FUNCTION_BLOCK SERVICE_INFO_JSON_DESERIALIZE (* Composite Function Block Type *)
  (* Standard: 61499-2 *)
  (* Version 0.0, 12/30/2022, brink, Flexbridge AB, template *)
  PACKAGE UAO.Hackathon;
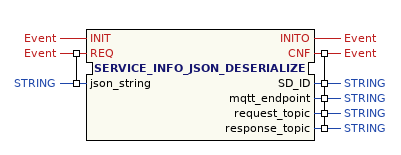
  EVENT_INPUT
    INIT;
    REQ WITH json_string; (* Normal Execution Request *)
  END_EVENT
  EVENT_OUTPUT
    INITO;
    CNF WITH SD_ID, mqtt_endpoint, request_topic, response_topic;
  END_EVENT
  VAR_INPUT
    json_string : STRING; (* Input event qualifier *)
  END_VAR
  VAR_OUTPUT
    SD_ID : STRING;
    mqtt_endpoint : STRING;
    request_topic : STRING;
    response_topic : STRING;
  END_VAR
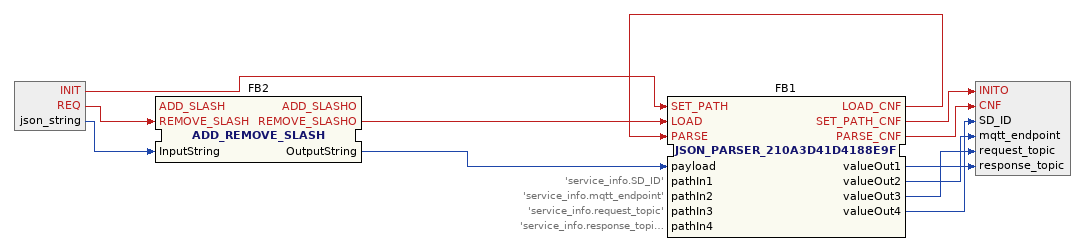
  FBS
    FB1 : JSON_PARSER_210A3D41D4188E9F(pathIn1 := 'service_info.SD_ID', pathIn2 := 'service_info.mqtt_endpoint', pathIn3 := 'service_info.request_topic', pathIn4 := 'service_info.response_topic'); {SET_ATTRIBUTE(Configuration.GenericFBType.InterfaceParams, Runtime.Base#CNT:=4;valueOut${CNT$}:STRING,STRING,STRING,STRING)}
    FB2 : ADD_REMOVE_SLASH;
  END_FBS
  EVENT_CONNECTIONS
    REQ TO FB2.REMOVE_SLASH;
    INIT TO FB1.SET_PATH;
    FB2.REMOVE_SLASHO TO FB1.LOAD;
    FB1.LOAD_CNF TO FB1.PARSE;
    FB1.SET_PATH_CNF TO INITO;
    FB1.PARSE_CNF TO CNF;
  END_CONNECTIONS
  DATA_CONNECTIONS
    json_string TO FB2.InputString;
    FB2.OutputString TO FB1.payload;
    FB1.valueOut1 TO SD_ID;
    FB1.valueOut2 TO mqtt_endpoint;
    FB1.valueOut3 TO request_topic;
    FB1.valueOut4 TO response_topic;
  END_CONNECTIONS
END_FUNCTION_BLOCK
